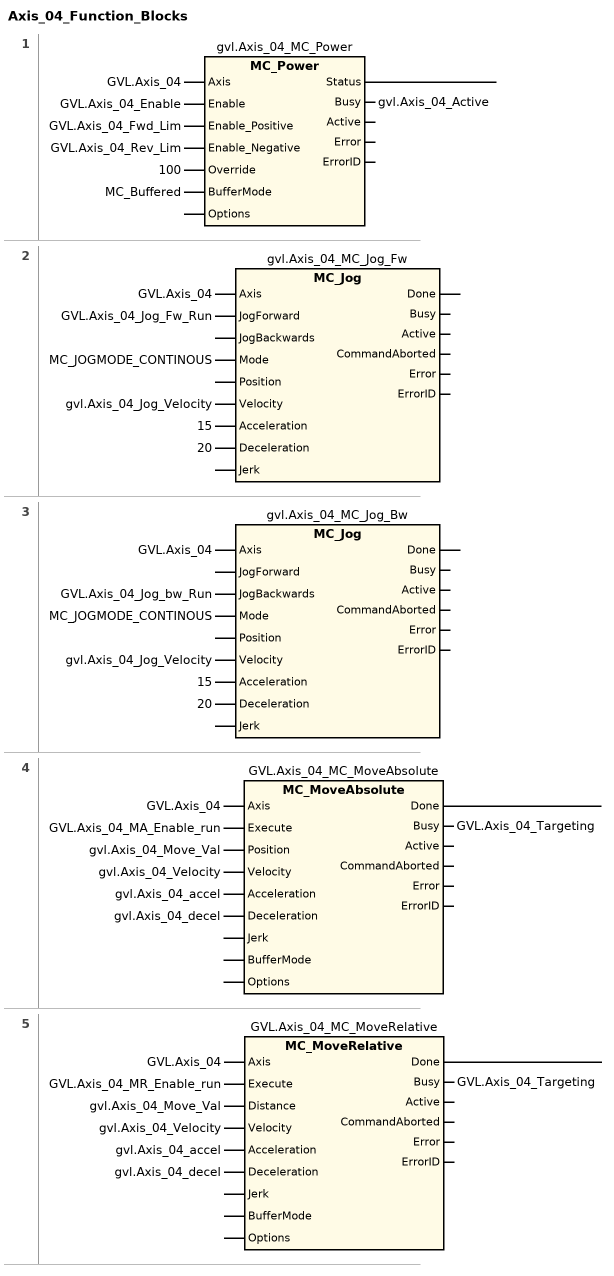
// NETWORK 1
gvl.Axis_04_MC_Power(
    Axis := GVL.Axis_04,
    Enable := GVL.Axis_04_Enable,
    Enable_Positive := GVL.Axis_04_Fwd_Lim,
    Enable_Negative := GVL.Axis_04_Rev_Lim,
    Override := 100,
    BufferMode := MC_Buffered,
    Busy => gvl.Axis_04_Active); // MC_Power

// NETWORK 2
gvl.Axis_04_MC_Jog_Fw(
    Axis := GVL.Axis_04,
    JogForward := GVL.Axis_04_Jog_Fw_Run,
    Mode := MC_JOGMODE_CONTINOUS,
    Velocity := gvl.Axis_04_Jog_Velocity,
    Acceleration := 15,
    Deceleration := 20); // MC_Jog

// NETWORK 3
gvl.Axis_04_MC_Jog_Bw(
    Axis := GVL.Axis_04,
    JogBackwards := GVL.Axis_04_Jog_bw_Run,
    Mode := MC_JOGMODE_CONTINOUS,
    Velocity := gvl.Axis_04_Jog_Velocity,
    Acceleration := 15,
    Deceleration := 20); // MC_Jog

// NETWORK 4
GVL.Axis_04_MC_MoveAbsolute(
    Axis := GVL.Axis_04,
    Execute := GVL.Axis_04_MA_Enable_run,
    Position := gvl.Axis_04_Move_Val,
    Velocity := gvl.Axis_04_Velocity,
    Acceleration := gvl.Axis_04_accel,
    Deceleration := gvl.Axis_04_decel,
    Busy => GVL.Axis_04_Targeting); // MC_MoveAbsolute

// NETWORK 5
GVL.Axis_04_MC_MoveRelative(
    Axis := GVL.Axis_04,
    Execute := GVL.Axis_04_MR_Enable_run,
    Distance := gvl.Axis_04_Move_Val,
    Velocity := gvl.Axis_04_Velocity,
    Acceleration := gvl.Axis_04_accel,
    Deceleration := gvl.Axis_04_decel,
    Busy => GVL.Axis_04_Targeting); // MC_MoveRelative

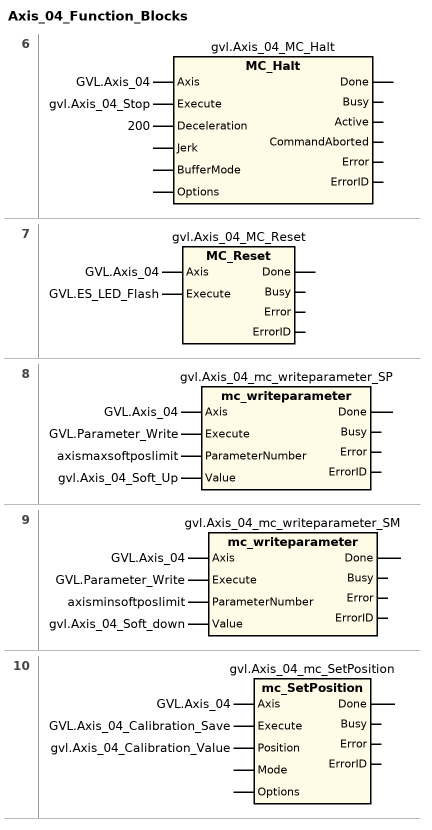
// NETWORK 6
gvl.Axis_04_MC_Halt(Axis := GVL.Axis_04, Execute := gvl.Axis_04_Stop, Deceleration := 200); // MC_Halt

// NETWORK 7
gvl.Axis_04_MC_Reset(Axis := GVL.Axis_04, Execute := GVL.ES_LED_Flash); // MC_Reset

// NETWORK 8
gvl.Axis_04_mc_writeparameter_SP(
    Axis := GVL.Axis_04,
    Execute := GVL.Parameter_Write,
    ParameterNumber := axismaxsoftposlimit,
    Value := gvl.Axis_04_Soft_Up); // mc_writeparameter

// NETWORK 9
gvl.Axis_04_mc_writeparameter_SM(
    Axis := GVL.Axis_04,
    Execute := GVL.Parameter_Write,
    ParameterNumber := axisminsoftposlimit,
    Value := gvl.Axis_04_Soft_down); // mc_writeparameter

// NETWORK 10
gvl.Axis_04_mc_SetPosition(
    Axis := GVL.Axis_04,
    Execute := GVL.Axis_04_Calibration_Save,
    Position := gvl.Axis_04_Calibration_Value); // mc_SetPosition

END_PROGRAM

// ---- POUs/Axis_04_Logic.TcPOU
PROGRAM Axis_04_Logic
VAR
	TON_0: TON;
	TON_1: TON;
	TON_2: TON;
	TON_3: TON;
	Axis_04_Velocity_Range: LREAL;
	Axis_04_Velocity_Scale: LREAL;
	Axis_04_Velocity_Raw: LREAL;
	Axis_04_Soft_Range: LREAL;
	Axis_04_Soft_Position: LREAL;
	Axis_04_Soft_Position_In_Range: LREAL;
END_VAR

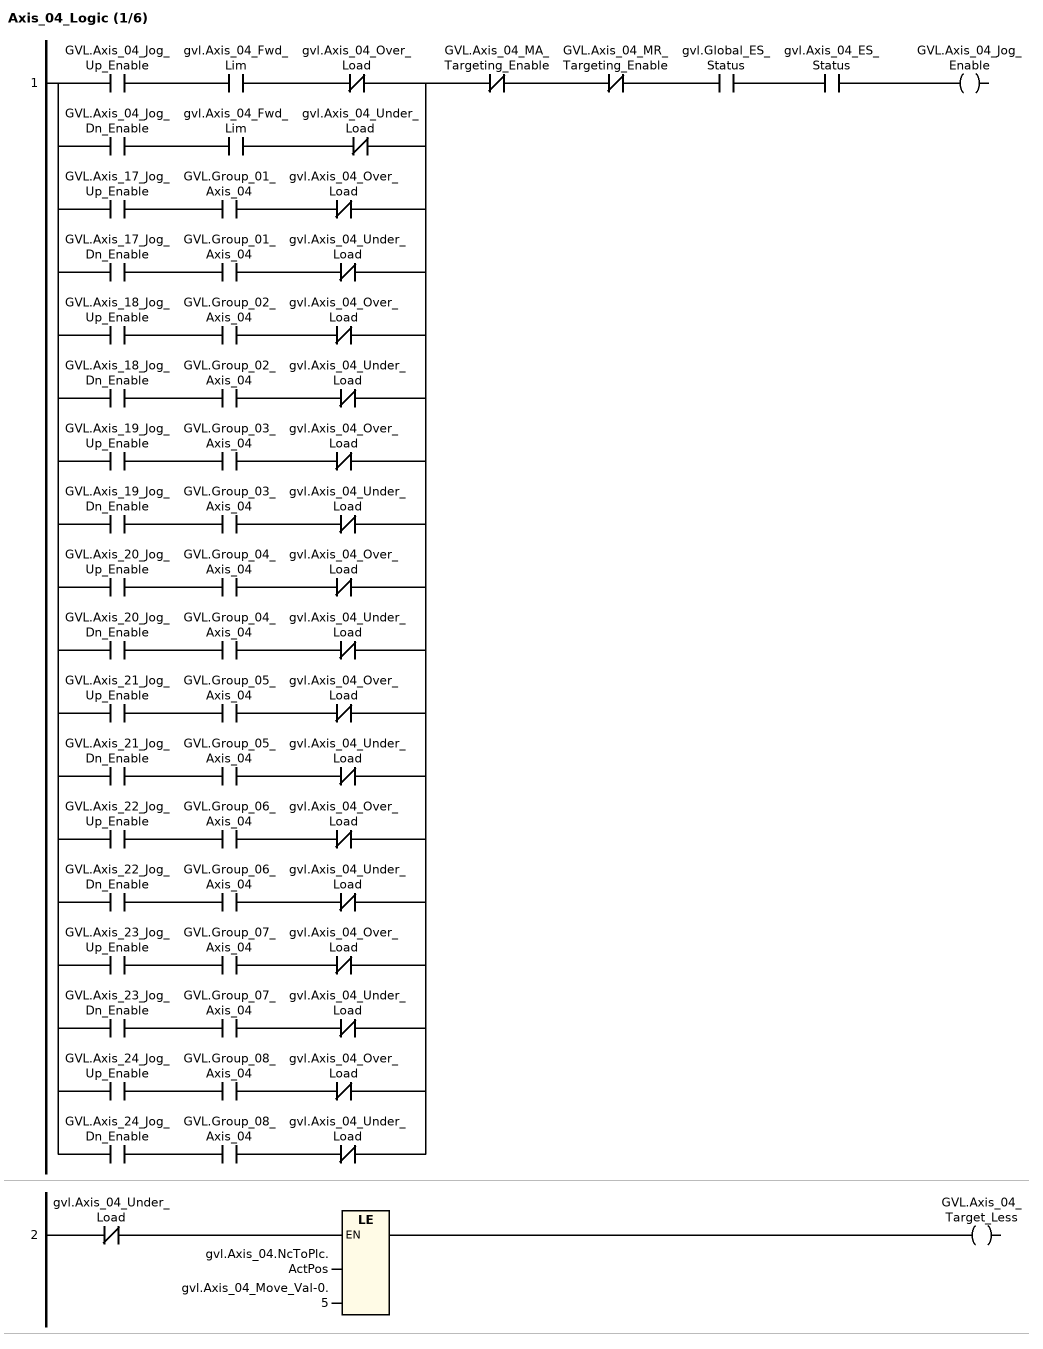
// NETWORK 1
GVL.Axis_04_Jog_Enable := (GVL.Axis_04_Jog_Up_Enable AND gvl.Axis_04_Fwd_Lim AND NOT gvl.Axis_04_Over_Load OR GVL.Axis_04_Jog_Dn_Enable AND gvl.Axis_04_Fwd_Lim AND NOT gvl.Axis_04_Under_Load OR GVL.Axis_17_Jog_Up_Enable AND GVL.Group_01_Axis_04 AND NOT gvl.Axis_04_Over_Load OR GVL.Axis_17_Jog_Dn_Enable AND GVL.Group_01_Axis_04 AND NOT gvl.Axis_04_Under_Load OR GVL.Axis_18_Jog_Up_Enable AND GVL.Group_02_Axis_04 AND NOT gvl.Axis_04_Over_Load OR GVL.Axis_18_Jog_Dn_Enable AND GVL.Group_02_Axis_04 AND NOT gvl.Axis_04_Under_Load OR GVL.Axis_19_Jog_Up_Enable AND GVL.Group_03_Axis_04 AND NOT gvl.Axis_04_Over_Load OR GVL.Axis_19_Jog_Dn_Enable AND GVL.Group_03_Axis_04 AND NOT gvl.Axis_04_Under_Load OR GVL.Axis_20_Jog_Up_Enable AND GVL.Group_04_Axis_04 AND NOT gvl.Axis_04_Over_Load OR GVL.Axis_20_Jog_Dn_Enable AND GVL.Group_04_Axis_04 AND NOT gvl.Axis_04_Under_Load OR GVL.Axis_21_Jog_Up_Enable AND GVL.Group_05_Axis_04 AND NOT gvl.Axis_04_Over_Load OR GVL.Axis_21_Jog_Dn_Enable AND GVL.Group_05_Axis_04 AND NOT gvl.Axis_04_Under_Load OR GVL.Axis_22_Jog_Up_Enable AND GVL.Group_06_Axis_04 AND NOT gvl.Axis_04_Over_Load OR GVL.Axis_22_Jog_Dn_Enable AND GVL.Group_06_Axis_04 AND NOT gvl.Axis_04_Under_Load OR GVL.Axis_23_Jog_Up_Enable AND GVL.Group_07_Axis_04 AND NOT gvl.Axis_04_Over_Load OR GVL.Axis_23_Jog_Dn_Enable AND GVL.Group_07_Axis_04 AND NOT gvl.Axis_04_Under_Load OR GVL.Axis_24_Jog_Up_Enable AND GVL.Group_08_Axis_04 AND NOT gvl.Axis_04_Over_Load OR GVL.Axis_24_Jog_Dn_Enable AND GVL.Group_08_Axis_04 AND NOT gvl.Axis_04_Under_Load) AND NOT GVL.Axis_04_MA_Targeting_Enable AND NOT GVL.Axis_04_MR_Targeting_Enable AND gvl.Global_ES_Status AND gvl.Axis_04_ES_Status;

// NETWORK 2
GVL.Axis_04_Target_Less := NOT gvl.Axis_04_Under_Load AND gvl.Axis_04.NcToPlc.ActPos <= (gvl.Axis_04_Move_Val-0.5);

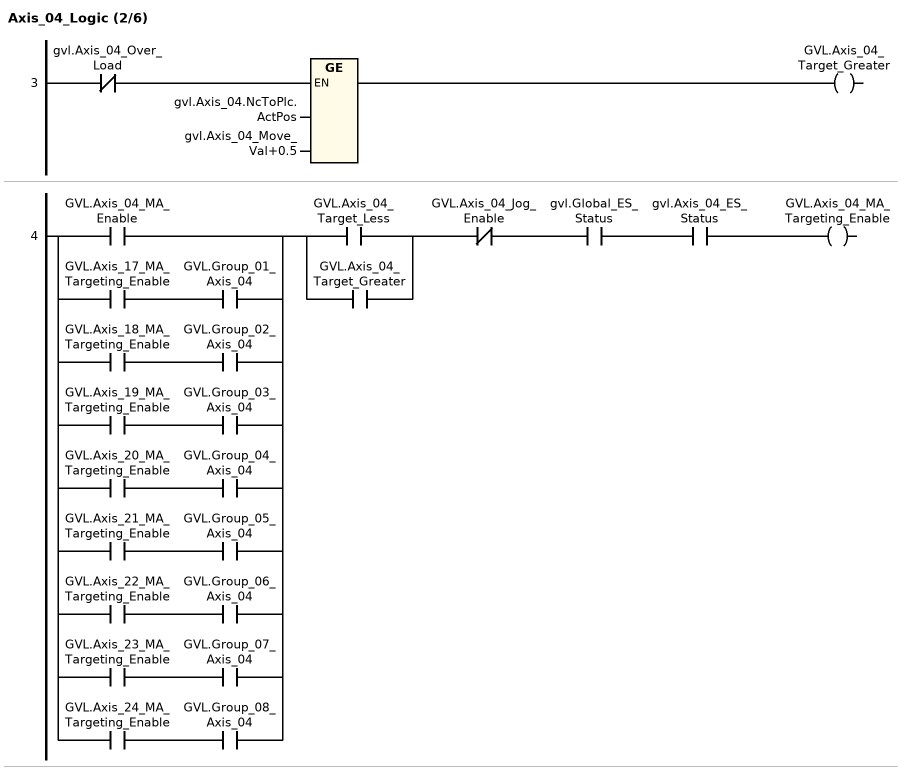
// NETWORK 3
GVL.Axis_04_Target_Greater := NOT gvl.Axis_04_Over_Load AND gvl.Axis_04.NcToPlc.ActPos >= (gvl.Axis_04_Move_Val+0.5);

// NETWORK 4
GVL.Axis_04_MA_Targeting_Enable := (GVL.Axis_04_MA_Enable OR GVL.Axis_17_MA_Targeting_Enable AND GVL.Group_01_Axis_04 OR GVL.Axis_18_MA_Targeting_Enable AND GVL.Group_02_Axis_04 OR GVL.Axis_19_MA_Targeting_Enable AND GVL.Group_03_Axis_04 OR GVL.Axis_20_MA_Targeting_Enable AND GVL.Group_04_Axis_04 OR GVL.Axis_21_MA_Targeting_Enable AND GVL.Group_05_Axis_04 OR GVL.Axis_22_MA_Targeting_Enable AND GVL.Group_06_Axis_04 OR GVL.Axis_23_MA_Targeting_Enable AND GVL.Group_07_Axis_04 OR GVL.Axis_24_MA_Targeting_Enable AND GVL.Group_08_Axis_04) AND (GVL.Axis_04_Target_Less OR GVL.Axis_04_Target_Greater) AND NOT GVL.Axis_04_Jog_Enable AND gvl.Global_ES_Status AND gvl.Axis_04_ES_Status;

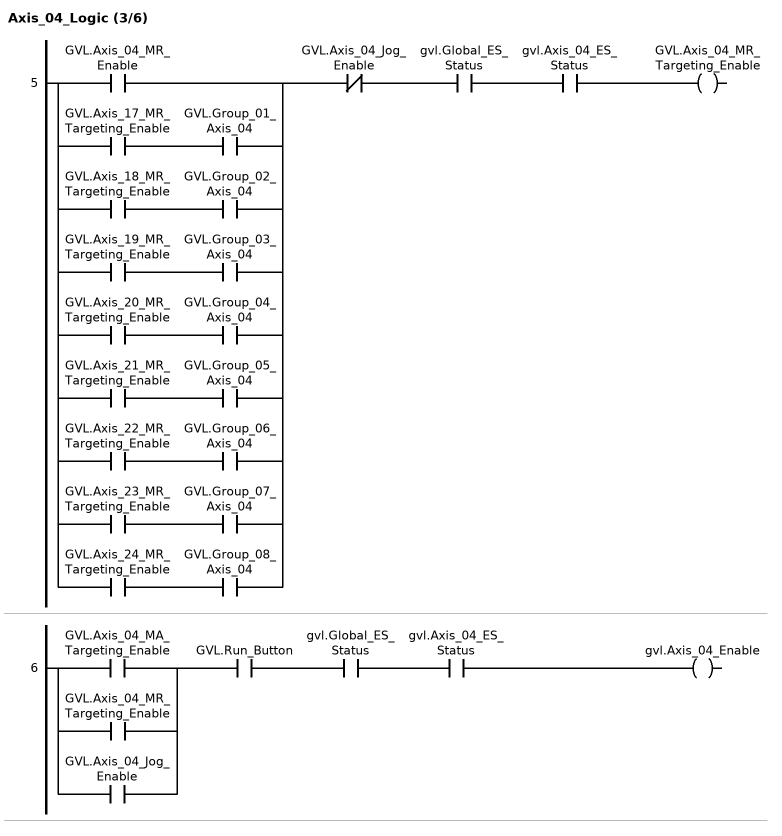
// NETWORK 5
GVL.Axis_04_MR_Targeting_Enable := (GVL.Axis_04_MR_Enable OR GVL.Axis_17_MR_Targeting_Enable AND GVL.Group_01_Axis_04 OR GVL.Axis_18_MR_Targeting_Enable AND GVL.Group_02_Axis_04 OR GVL.Axis_19_MR_Targeting_Enable AND GVL.Group_03_Axis_04 OR GVL.Axis_20_MR_Targeting_Enable AND GVL.Group_04_Axis_04 OR GVL.Axis_21_MR_Targeting_Enable AND GVL.Group_05_Axis_04 OR GVL.Axis_22_MR_Targeting_Enable AND GVL.Group_06_Axis_04 OR GVL.Axis_23_MR_Targeting_Enable AND GVL.Group_07_Axis_04 OR GVL.Axis_24_MR_Targeting_Enable AND GVL.Group_08_Axis_04) AND NOT GVL.Axis_04_Jog_Enable AND gvl.Global_ES_Status AND gvl.Axis_04_ES_Status;

// NETWORK 6
gvl.Axis_04_Enable := (GVL.Axis_04_MA_Targeting_Enable OR GVL.Axis_04_MR_Targeting_Enable OR GVL.Axis_04_Jog_Enable) AND GVL.Run_Button AND gvl.Global_ES_Status AND gvl.Axis_04_ES_Status;

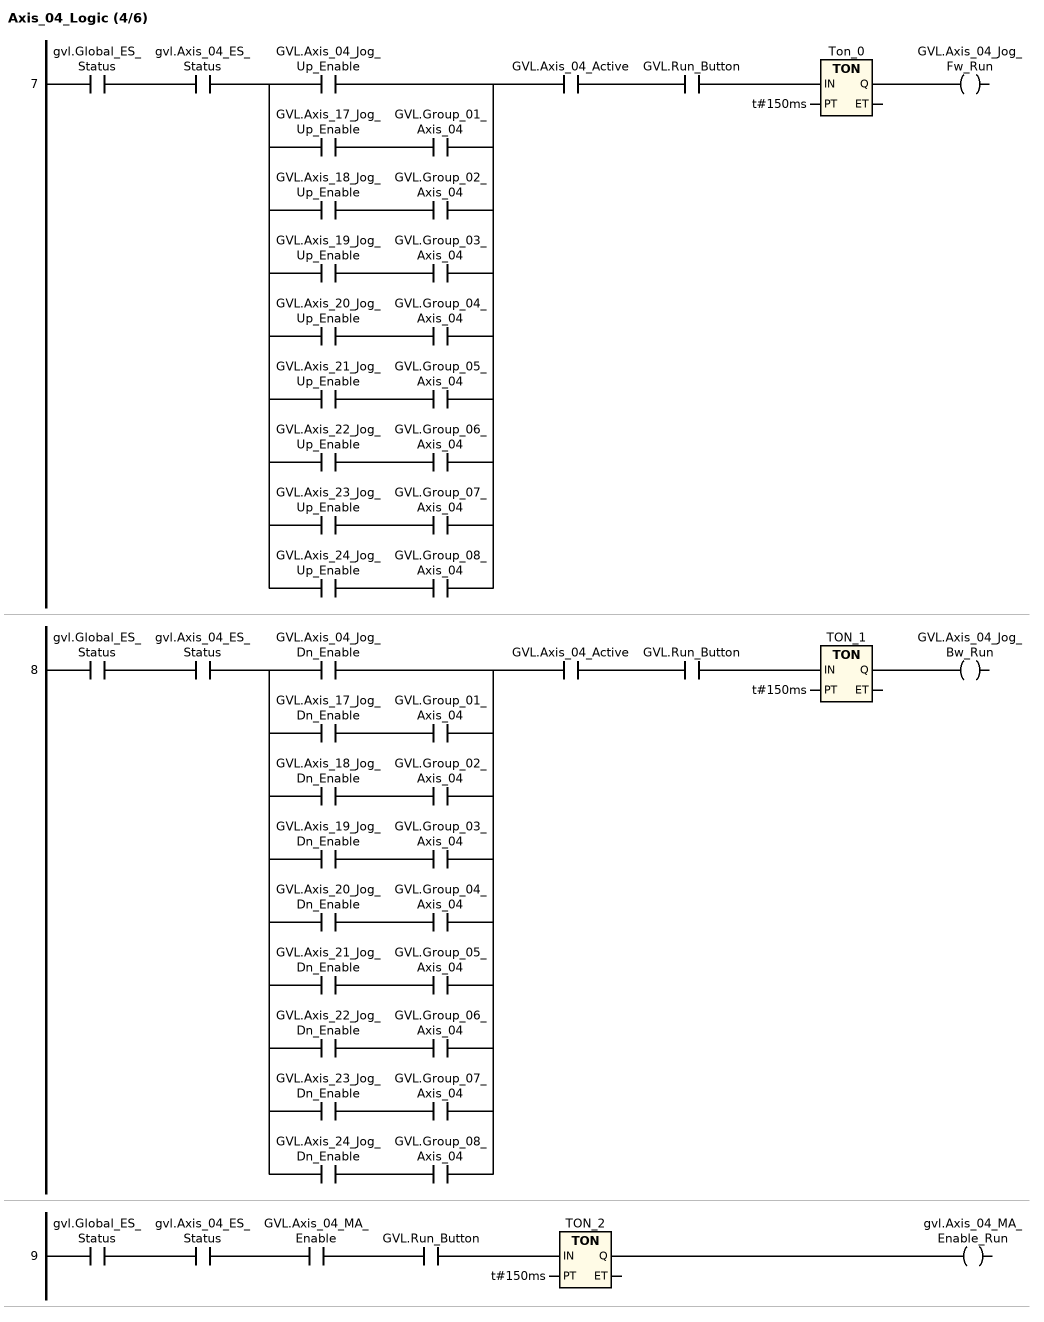
// NETWORK 7
Ton_0(IN := gvl.Global_ES_Status AND gvl.Axis_04_ES_Status AND (GVL.Axis_04_Jog_Up_Enable OR GVL.Axis_17_Jog_Up_Enable AND GVL.Group_01_Axis_04 OR GVL.Axis_18_Jog_Up_Enable AND GVL.Group_02_Axis_04 OR GVL.Axis_19_Jog_Up_Enable AND GVL.Group_03_Axis_04 OR GVL.Axis_20_Jog_Up_Enable AND GVL.Group_04_Axis_04 OR GVL.Axis_21_Jog_Up_Enable AND GVL.Group_05_Axis_04 OR GVL.Axis_22_Jog_Up_Enable AND GVL.Group_06_Axis_04 OR GVL.Axis_23_Jog_Up_Enable AND GVL.Group_07_Axis_04 OR GVL.Axis_24_Jog_Up_Enable AND GVL.Group_08_Axis_04) AND GVL.Axis_04_Active AND GVL.Run_Button, PT := t#150ms); // TON
GVL.Axis_04_Jog_Fw_Run := Ton_0.Q;

// NETWORK 8
TON_1(IN := gvl.Global_ES_Status AND gvl.Axis_04_ES_Status AND (GVL.Axis_04_Jog_Dn_Enable OR GVL.Axis_17_Jog_Dn_Enable AND GVL.Group_01_Axis_04 OR GVL.Axis_18_Jog_Dn_Enable AND GVL.Group_02_Axis_04 OR GVL.Axis_19_Jog_Dn_Enable AND GVL.Group_03_Axis_04 OR GVL.Axis_20_Jog_Dn_Enable AND GVL.Group_04_Axis_04 OR GVL.Axis_21_Jog_Dn_Enable AND GVL.Group_05_Axis_04 OR GVL.Axis_22_Jog_Dn_Enable AND GVL.Group_06_Axis_04 OR GVL.Axis_23_Jog_Dn_Enable AND GVL.Group_07_Axis_04 OR GVL.Axis_24_Jog_Dn_Enable AND GVL.Group_08_Axis_04) AND GVL.Axis_04_Active AND GVL.Run_Button, PT := t#150ms); // TON
GVL.Axis_04_Jog_Bw_Run := TON_1.Q;

// NETWORK 9
TON_2(IN := gvl.Global_ES_Status AND gvl.Axis_04_ES_Status AND GVL.Axis_04_MA_Enable AND GVL.Run_Button, PT := t#150ms); // TON
gvl.Axis_04_MA_Enable_Run := TON_2.Q;

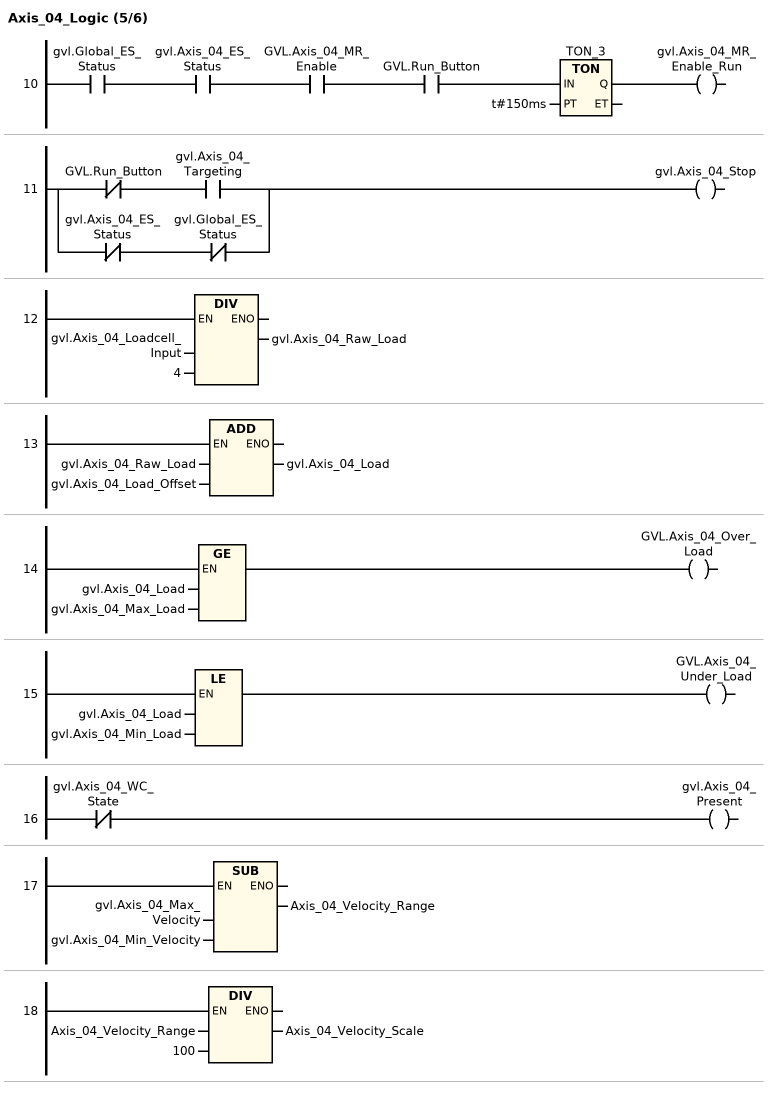
// NETWORK 10
TON_3(IN := gvl.Global_ES_Status AND gvl.Axis_04_ES_Status AND GVL.Axis_04_MR_Enable AND GVL.Run_Button, PT := t#150ms); // TON
gvl.Axis_04_MR_Enable_Run := TON_3.Q;

// NETWORK 11
gvl.Axis_04_Stop := NOT GVL.Run_Button AND gvl.Axis_04_Targeting OR NOT gvl.Axis_04_ES_Status AND NOT gvl.Global_ES_Status;

// NETWORK 12
gvl.Axis_04_Raw_Load := gvl.Axis_04_Loadcell_Input / 4;

// NETWORK 13
gvl.Axis_04_Load := gvl.Axis_04_Raw_Load + gvl.Axis_04_Load_Offset;

// NETWORK 14
GVL.Axis_04_Over_Load := gvl.Axis_04_Load >= gvl.Axis_04_Max_Load;

// NETWORK 15
GVL.Axis_04_Under_Load := gvl.Axis_04_Load <= gvl.Axis_04_Min_Load;

// NETWORK 16
gvl.Axis_04_Present := NOT gvl.Axis_04_WC_State;

// NETWORK 17
Axis_04_Velocity_Range := gvl.Axis_04_Max_Velocity - gvl.Axis_04_Min_Velocity;

// NETWORK 18
Axis_04_Velocity_Scale := Axis_04_Velocity_Range / 100;

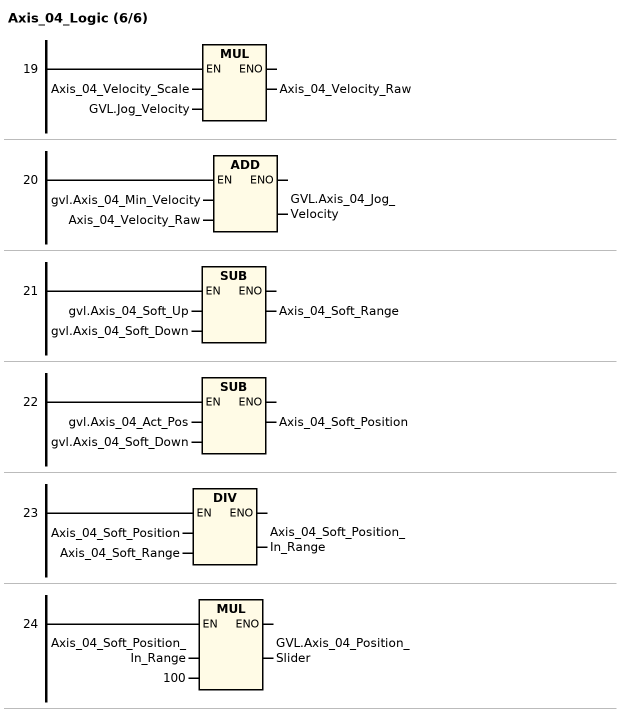
// NETWORK 19
Axis_04_Velocity_Raw := Axis_04_Velocity_Scale * GVL.Jog_Velocity;

// NETWORK 20
GVL.Axis_04_Jog_Velocity := gvl.Axis_04_Min_Velocity + Axis_04_Velocity_Raw;

// NETWORK 21
Axis_04_Soft_Range := gvl.Axis_04_Soft_Up - gvl.Axis_04_Soft_Down;

// NETWORK 22
Axis_04_Soft_Position := gvl.Axis_04_Act_Pos - gvl.Axis_04_Soft_Down;

// NETWORK 23
Axis_04_Soft_Position_In_Range := Axis_04_Soft_Position / Axis_04_Soft_Range;

// NETWORK 24
GVL.Axis_04_Position_Slider := Axis_04_Soft_Position_In_Range * 100;

END_PROGRAM

// ---- POUs/Axis_05_Function_Blocks.TcPOU
PROGRAM Axis_05_Function_Blocks
VAR
END_VAR

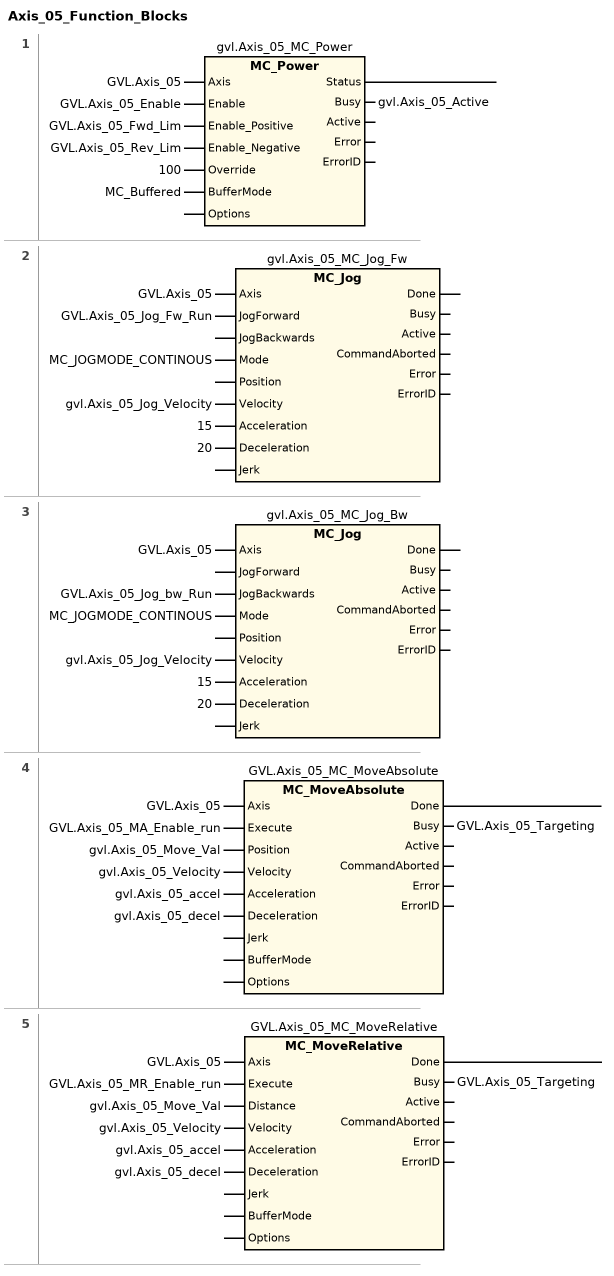
// NETWORK 1
gvl.Axis_05_MC_Power(
    Axis := GVL.Axis_05,
    Enable := GVL.Axis_05_Enable,
    Enable_Positive := GVL.Axis_05_Fwd_Lim,
    Enable_Negative := GVL.Axis_05_Rev_Lim,
    Override := 100,
    BufferMode := MC_Buffered,
    Busy => gvl.Axis_05_Active); // MC_Power

// NETWORK 2
gvl.Axis_05_MC_Jog_Fw(
    Axis := GVL.Axis_05,
    JogForward := GVL.Axis_05_Jog_Fw_Run,
    Mode := MC_JOGMODE_CONTINOUS,
    Velocity := gvl.Axis_05_Jog_Velocity,
    Acceleration := 15,
    Deceleration := 20); // MC_Jog

// NETWORK 3
gvl.Axis_05_MC_Jog_Bw(
    Axis := GVL.Axis_05,
    JogBackwards := GVL.Axis_05_Jog_bw_Run,
    Mode := MC_JOGMODE_CONTINOUS,
    Velocity := gvl.Axis_05_Jog_Velocity,
    Acceleration := 15,
    Deceleration := 20); // MC_Jog

// NETWORK 4
GVL.Axis_05_MC_MoveAbsolute(
    Axis := GVL.Axis_05,
    Execute := GVL.Axis_05_MA_Enable_run,
    Position := gvl.Axis_05_Move_Val,
    Velocity := gvl.Axis_05_Velocity,
    Acceleration := gvl.Axis_05_accel,
    Deceleration := gvl.Axis_05_decel,
    Busy => GVL.Axis_05_Targeting); // MC_MoveAbsolute

// NETWORK 5
GVL.Axis_05_MC_MoveRelative(
    Axis := GVL.Axis_05,
    Execute := GVL.Axis_05_MR_Enable_run,
    Distance := gvl.Axis_05_Move_Val,
    Velocity := gvl.Axis_05_Velocity,
    Acceleration := gvl.Axis_05_accel,
    Deceleration := gvl.Axis_05_decel,
    Busy => GVL.Axis_05_Targeting); // MC_MoveRelative

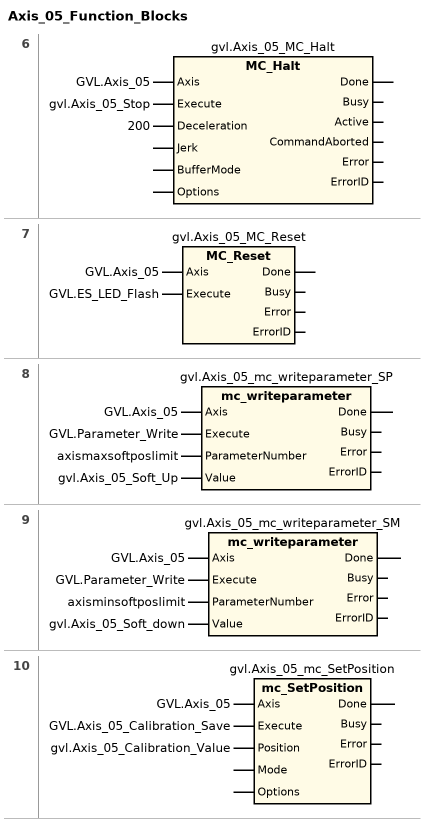
// NETWORK 6
gvl.Axis_05_MC_Halt(Axis := GVL.Axis_05, Execute := gvl.Axis_05_Stop, Deceleration := 200); // MC_Halt

// NETWORK 7
gvl.Axis_05_MC_Reset(Axis := GVL.Axis_05, Execute := GVL.ES_LED_Flash); // MC_Reset

// NETWORK 8
gvl.Axis_05_mc_writeparameter_SP(
    Axis := GVL.Axis_05,
    Execute := GVL.Parameter_Write,
    ParameterNumber := axismaxsoftposlimit,
    Value := gvl.Axis_05_Soft_Up); // mc_writeparameter

// NETWORK 9
gvl.Axis_05_mc_writeparameter_SM(
    Axis := GVL.Axis_05,
    Execute := GVL.Parameter_Write,
    ParameterNumber := axisminsoftposlimit,
    Value := gvl.Axis_05_Soft_down); // mc_writeparameter

// NETWORK 10
gvl.Axis_05_mc_SetPosition(
    Axis := GVL.Axis_05,
    Execute := GVL.Axis_05_Calibration_Save,
    Position := gvl.Axis_05_Calibration_Value); // mc_SetPosition

END_PROGRAM

// ---- POUs/Axis_05_Logic.TcPOU
PROGRAM Axis_05_Logic
VAR
	TON_0: TON;
	TON_1: TON;
	TON_2: TON;
	TON_3: TON;
	Axis_05_Velocity_Range: LREAL;
	Axis_05_Velocity_Scale: LREAL;
	Axis_05_Velocity_Raw: LREAL;
	Axis_05_Soft_Range: LREAL;
	Axis_05_Soft_Position: LREAL;
	Axis_05_Soft_Position_In_Range: LREAL;
END_VAR

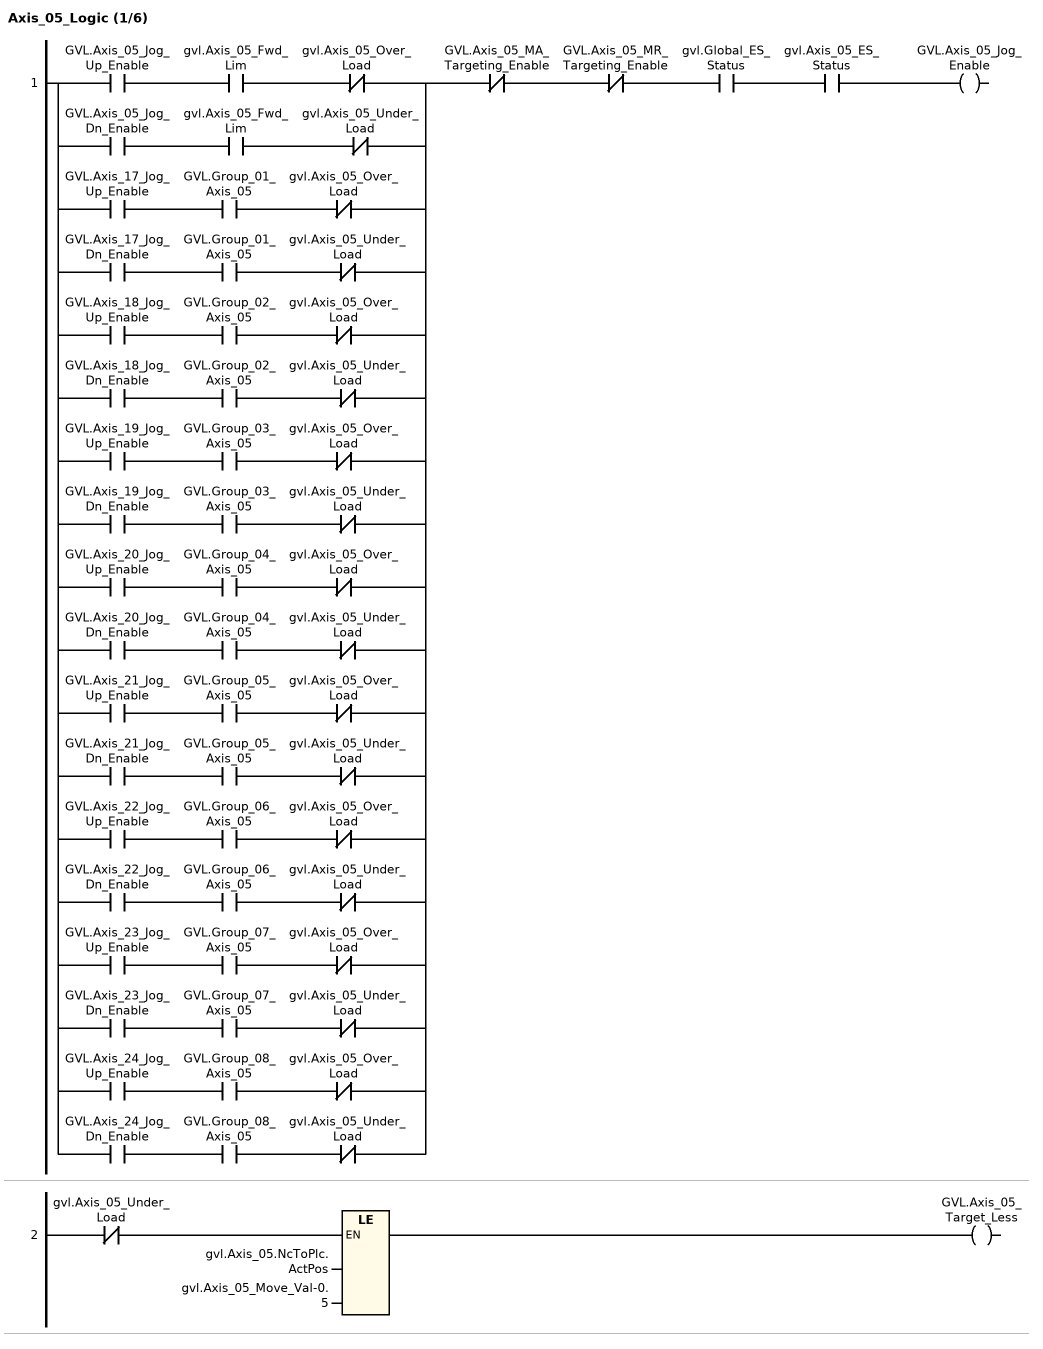
// NETWORK 1
GVL.Axis_05_Jog_Enable := (GVL.Axis_05_Jog_Up_Enable AND gvl.Axis_05_Fwd_Lim AND NOT gvl.Axis_05_Over_Load OR GVL.Axis_05_Jog_Dn_Enable AND gvl.Axis_05_Fwd_Lim AND NOT gvl.Axis_05_Under_Load OR GVL.Axis_17_Jog_Up_Enable AND GVL.Group_01_Axis_05 AND NOT gvl.Axis_05_Over_Load OR GVL.Axis_17_Jog_Dn_Enable AND GVL.Group_01_Axis_05 AND NOT gvl.Axis_05_Under_Load OR GVL.Axis_18_Jog_Up_Enable AND GVL.Group_02_Axis_05 AND NOT gvl.Axis_05_Over_Load OR GVL.Axis_18_Jog_Dn_Enable AND GVL.Group_02_Axis_05 AND NOT gvl.Axis_05_Under_Load OR GVL.Axis_19_Jog_Up_Enable AND GVL.Group_03_Axis_05 AND NOT gvl.Axis_05_Over_Load OR GVL.Axis_19_Jog_Dn_Enable AND GVL.Group_03_Axis_05 AND NOT gvl.Axis_05_Under_Load OR GVL.Axis_20_Jog_Up_Enable AND GVL.Group_04_Axis_05 AND NOT gvl.Axis_05_Over_Load OR GVL.Axis_20_Jog_Dn_Enable AND GVL.Group_04_Axis_05 AND NOT gvl.Axis_05_Under_Load OR GVL.Axis_21_Jog_Up_Enable AND GVL.Group_05_Axis_05 AND NOT gvl.Axis_05_Over_Load OR GVL.Axis_21_Jog_Dn_Enable AND GVL.Group_05_Axis_05 AND NOT gvl.Axis_05_Under_Load OR GVL.Axis_22_Jog_Up_Enable AND GVL.Group_06_Axis_05 AND NOT gvl.Axis_05_Over_Load OR GVL.Axis_22_Jog_Dn_Enable AND GVL.Group_06_Axis_05 AND NOT gvl.Axis_05_Under_Load OR GVL.Axis_23_Jog_Up_Enable AND GVL.Group_07_Axis_05 AND NOT gvl.Axis_05_Over_Load OR GVL.Axis_23_Jog_Dn_Enable AND GVL.Group_07_Axis_05 AND NOT gvl.Axis_05_Under_Load OR GVL.Axis_24_Jog_Up_Enable AND GVL.Group_08_Axis_05 AND NOT gvl.Axis_05_Over_Load OR GVL.Axis_24_Jog_Dn_Enable AND GVL.Group_08_Axis_05 AND NOT gvl.Axis_05_Under_Load) AND NOT GVL.Axis_05_MA_Targeting_Enable AND NOT GVL.Axis_05_MR_Targeting_Enable AND gvl.Global_ES_Status AND gvl.Axis_05_ES_Status;

// NETWORK 2
GVL.Axis_05_Target_Less := NOT gvl.Axis_05_Under_Load AND gvl.Axis_05.NcToPlc.ActPos <= (gvl.Axis_05_Move_Val-0.5);

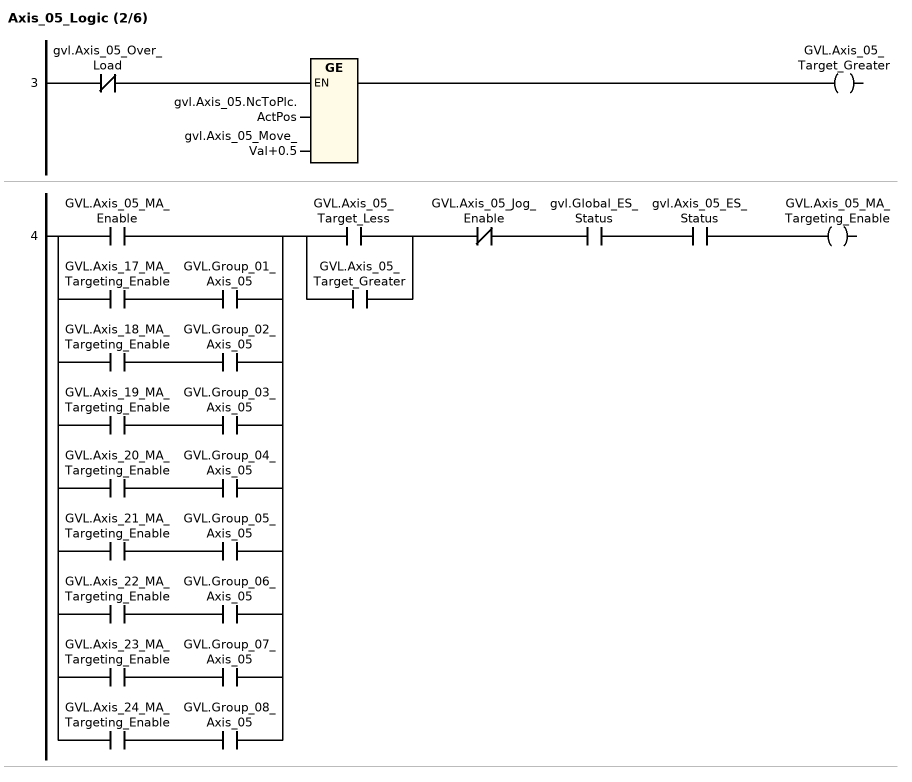
// NETWORK 3
GVL.Axis_05_Target_Greater := NOT gvl.Axis_05_Over_Load AND gvl.Axis_05.NcToPlc.ActPos >= (gvl.Axis_05_Move_Val+0.5);

// NETWORK 4
GVL.Axis_05_MA_Targeting_Enable := (GVL.Axis_05_MA_Enable OR GVL.Axis_17_MA_Targeting_Enable AND GVL.Group_01_Axis_05 OR GVL.Axis_18_MA_Targeting_Enable AND GVL.Group_02_Axis_05 OR GVL.Axis_19_MA_Targeting_Enable AND GVL.Group_03_Axis_05 OR GVL.Axis_20_MA_Targeting_Enable AND GVL.Group_04_Axis_05 OR GVL.Axis_21_MA_Targeting_Enable AND GVL.Group_05_Axis_05 OR GVL.Axis_22_MA_Targeting_Enable AND GVL.Group_06_Axis_05 OR GVL.Axis_23_MA_Targeting_Enable AND GVL.Group_07_Axis_05 OR GVL.Axis_24_MA_Targeting_Enable AND GVL.Group_08_Axis_05) AND (GVL.Axis_05_Target_Less OR GVL.Axis_05_Target_Greater) AND NOT GVL.Axis_05_Jog_Enable AND gvl.Global_ES_Status AND gvl.Axis_05_ES_Status;

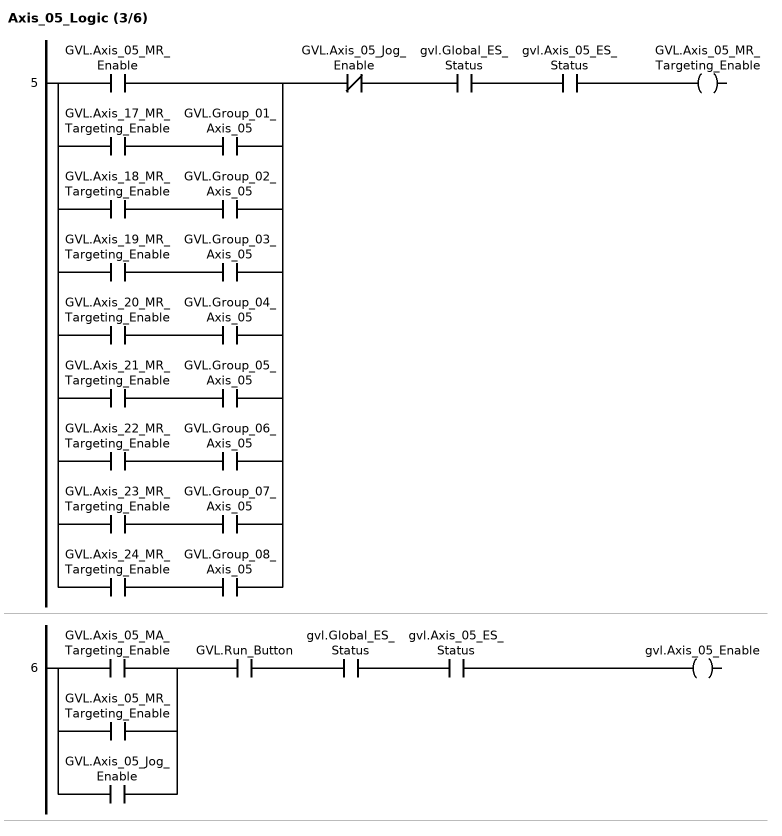
// NETWORK 5
GVL.Axis_05_MR_Targeting_Enable := (GVL.Axis_05_MR_Enable OR GVL.Axis_17_MR_Targeting_Enable AND GVL.Group_01_Axis_05 OR GVL.Axis_18_MR_Targeting_Enable AND GVL.Group_02_Axis_05 OR GVL.Axis_19_MR_Targeting_Enable AND GVL.Group_03_Axis_05 OR GVL.Axis_20_MR_Targeting_Enable AND GVL.Group_04_Axis_05 OR GVL.Axis_21_MR_Targeting_Enable AND GVL.Group_05_Axis_05 OR GVL.Axis_22_MR_Targeting_Enable AND GVL.Group_06_Axis_05 OR GVL.Axis_23_MR_Targeting_Enable AND GVL.Group_07_Axis_05 OR GVL.Axis_24_MR_Targeting_Enable AND GVL.Group_08_Axis_05) AND NOT GVL.Axis_05_Jog_Enable AND gvl.Global_ES_Status AND gvl.Axis_05_ES_Status;

// NETWORK 6
gvl.Axis_05_Enable := (GVL.Axis_05_MA_Targeting_Enable OR GVL.Axis_05_MR_Targeting_Enable OR GVL.Axis_05_Jog_Enable) AND GVL.Run_Button AND gvl.Global_ES_Status AND gvl.Axis_05_ES_Status;

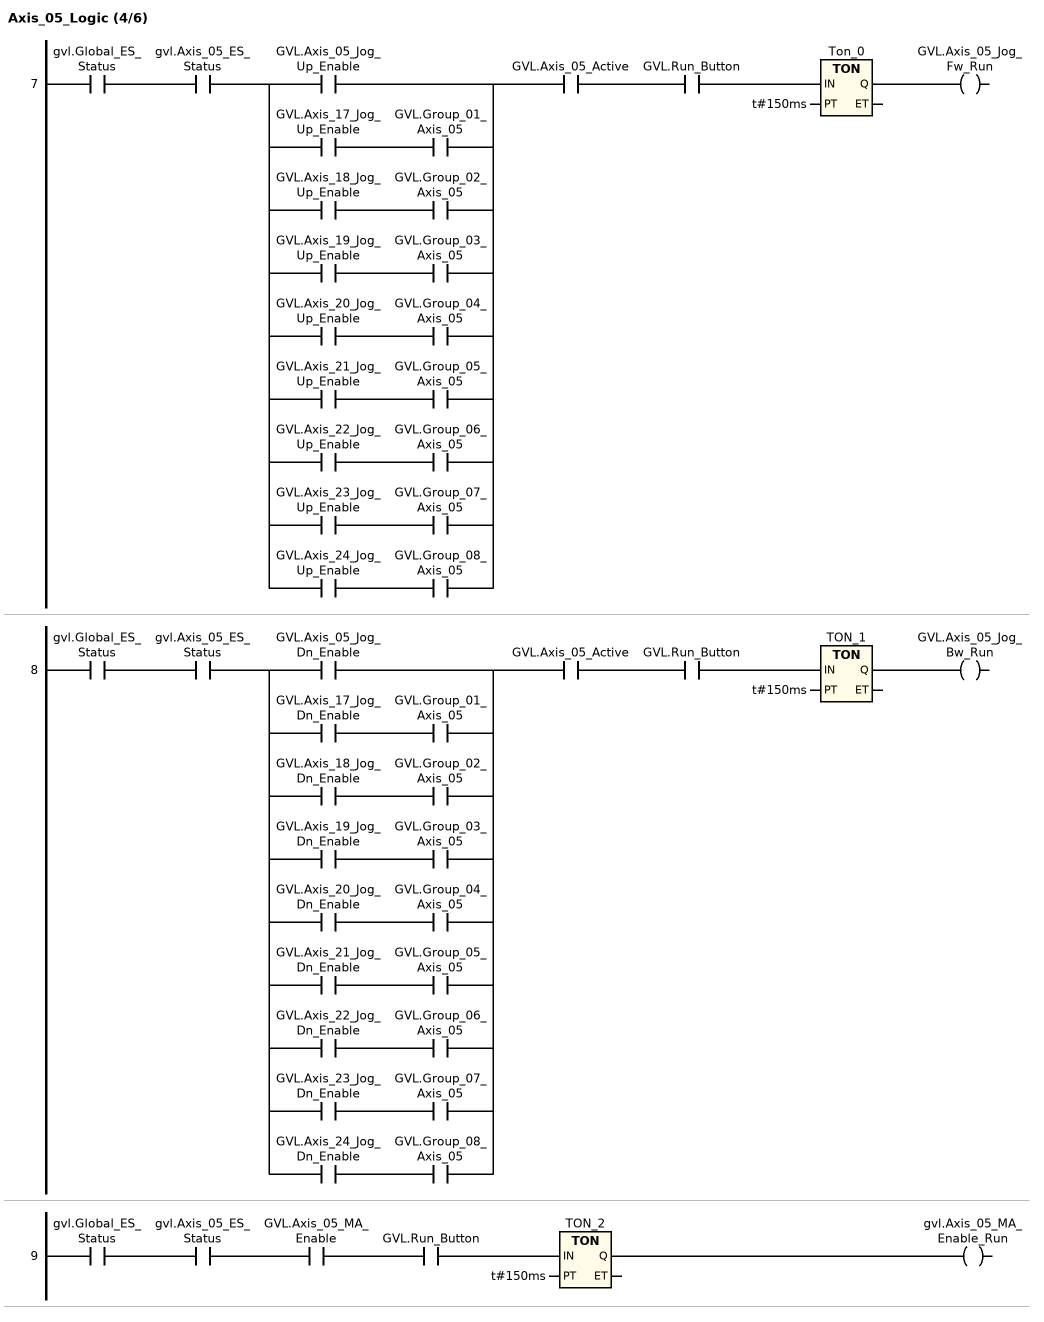
// NETWORK 7
Ton_0(IN := gvl.Global_ES_Status AND gvl.Axis_05_ES_Status AND (GVL.Axis_05_Jog_Up_Enable OR GVL.Axis_17_Jog_Up_Enable AND GVL.Group_01_Axis_05 OR GVL.Axis_18_Jog_Up_Enable AND GVL.Group_02_Axis_05 OR GVL.Axis_19_Jog_Up_Enable AND GVL.Group_03_Axis_05 OR GVL.Axis_20_Jog_Up_Enable AND GVL.Group_04_Axis_05 OR GVL.Axis_21_Jog_Up_Enable AND GVL.Group_05_Axis_05 OR GVL.Axis_22_Jog_Up_Enable AND GVL.Group_06_Axis_05 OR GVL.Axis_23_Jog_Up_Enable AND GVL.Group_07_Axis_05 OR GVL.Axis_24_Jog_Up_Enable AND GVL.Group_08_Axis_05) AND GVL.Axis_05_Active AND GVL.Run_Button, PT := t#150ms); // TON
GVL.Axis_05_Jog_Fw_Run := Ton_0.Q;

// NETWORK 8
TON_1(IN := gvl.Global_ES_Status AND gvl.Axis_05_ES_Status AND (GVL.Axis_05_Jog_Dn_Enable OR GVL.Axis_17_Jog_Dn_Enable AND GVL.Group_01_Axis_05 OR GVL.Axis_18_Jog_Dn_Enable AND GVL.Group_02_Axis_05 OR GVL.Axis_19_Jog_Dn_Enable AND GVL.Group_03_Axis_05 OR GVL.Axis_20_Jog_Dn_Enable AND GVL.Group_04_Axis_05 OR GVL.Axis_21_Jog_Dn_Enable AND GVL.Group_05_Axis_05 OR GVL.Axis_22_Jog_Dn_Enable AND GVL.Group_06_Axis_05 OR GVL.Axis_23_Jog_Dn_Enable AND GVL.Group_07_Axis_05 OR GVL.Axis_24_Jog_Dn_Enable AND GVL.Group_08_Axis_05) AND GVL.Axis_05_Active AND GVL.Run_Button, PT := t#150ms); // TON
GVL.Axis_05_Jog_Bw_Run := TON_1.Q;

// NETWORK 9
TON_2(IN := gvl.Global_ES_Status AND gvl.Axis_05_ES_Status AND GVL.Axis_05_MA_Enable AND GVL.Run_Button, PT := t#150ms); // TON
gvl.Axis_05_MA_Enable_Run := TON_2.Q;

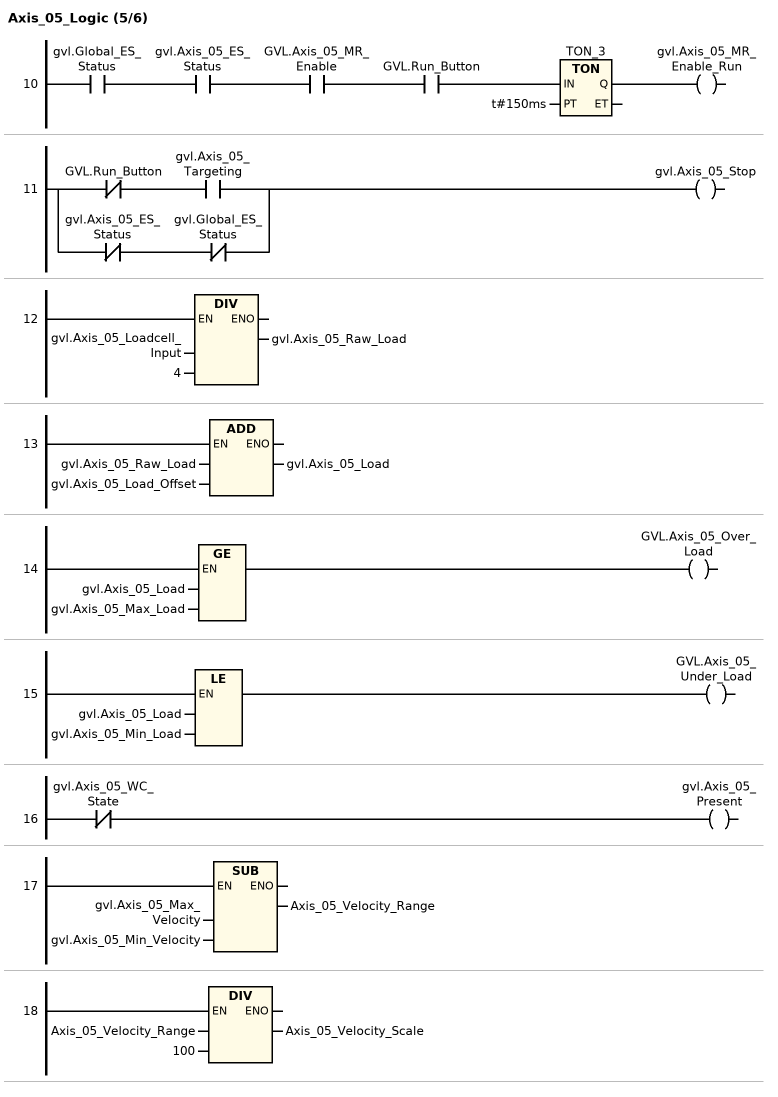
// NETWORK 10
TON_3(IN := gvl.Global_ES_Status AND gvl.Axis_05_ES_Status AND GVL.Axis_05_MR_Enable AND GVL.Run_Button, PT := t#150ms); // TON
gvl.Axis_05_MR_Enable_Run := TON_3.Q;

// NETWORK 11
gvl.Axis_05_Stop := NOT GVL.Run_Button AND gvl.Axis_05_Targeting OR NOT gvl.Axis_05_ES_Status AND NOT gvl.Global_ES_Status;

// NETWORK 12
gvl.Axis_05_Raw_Load := gvl.Axis_05_Loadcell_Input / 4;

// NETWORK 13
gvl.Axis_05_Load := gvl.Axis_05_Raw_Load + gvl.Axis_05_Load_Offset;

// NETWORK 14
GVL.Axis_05_Over_Load := gvl.Axis_05_Load >= gvl.Axis_05_Max_Load;

// NETWORK 15
GVL.Axis_05_Under_Load := gvl.Axis_05_Load <= gvl.Axis_05_Min_Load;

// NETWORK 16
gvl.Axis_05_Present := NOT gvl.Axis_05_WC_State;

// NETWORK 17
Axis_05_Velocity_Range := gvl.Axis_05_Max_Velocity - gvl.Axis_05_Min_Velocity;

// NETWORK 18
Axis_05_Velocity_Scale := Axis_05_Velocity_Range / 100;

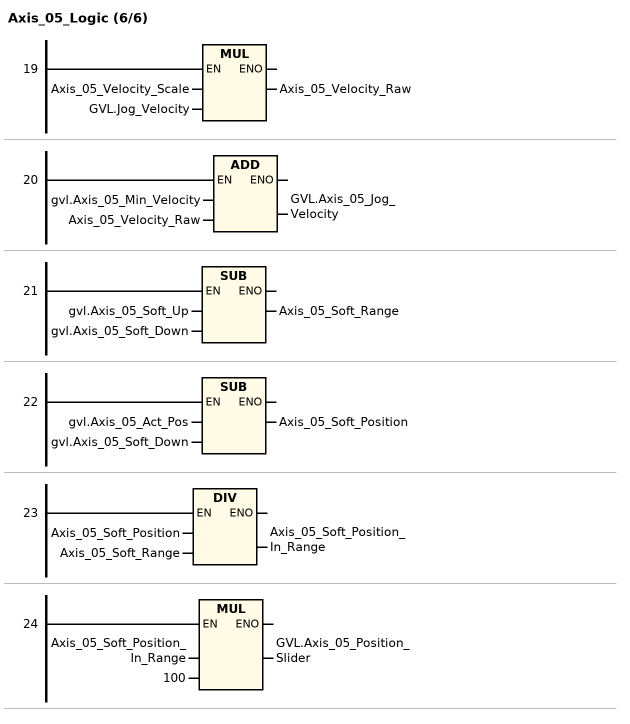
// NETWORK 19
Axis_05_Velocity_Raw := Axis_05_Velocity_Scale * GVL.Jog_Velocity;

// NETWORK 20
GVL.Axis_05_Jog_Velocity := gvl.Axis_05_Min_Velocity + Axis_05_Velocity_Raw;

// NETWORK 21
Axis_05_Soft_Range := gvl.Axis_05_Soft_Up - gvl.Axis_05_Soft_Down;

// NETWORK 22
Axis_05_Soft_Position := gvl.Axis_05_Act_Pos - gvl.Axis_05_Soft_Down;

// NETWORK 23
Axis_05_Soft_Position_In_Range := Axis_05_Soft_Position / Axis_05_Soft_Range;

// NETWORK 24
GVL.Axis_05_Position_Slider := Axis_05_Soft_Position_In_Range * 100;

END_PROGRAM

// ---- POUs/Axis_06_Function_Blocks.TcPOU
PROGRAM Axis_06_Function_Blocks
VAR
END_VAR

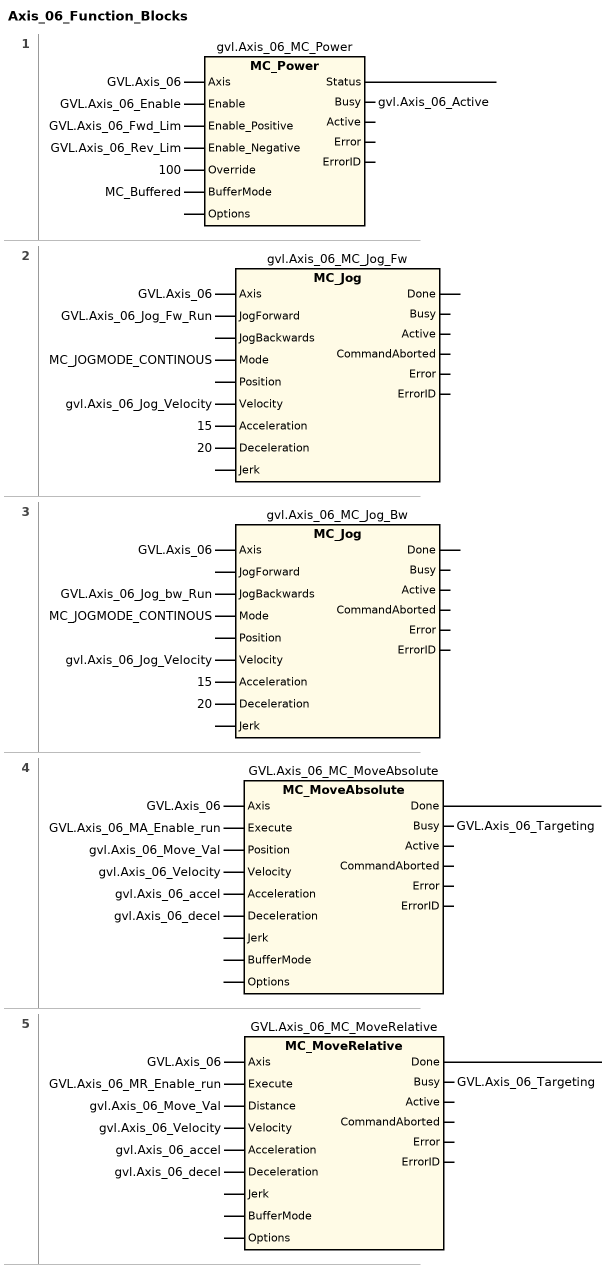
// NETWORK 1
gvl.Axis_06_MC_Power(
    Axis := GVL.Axis_06,
    Enable := GVL.Axis_06_Enable,
    Enable_Positive := GVL.Axis_06_Fwd_Lim,
    Enable_Negative := GVL.Axis_06_Rev_Lim,
    Override := 100,
    BufferMode := MC_Buffered,
    Busy => gvl.Axis_06_Active); // MC_Power

// NETWORK 2
gvl.Axis_06_MC_Jog_Fw(
    Axis := GVL.Axis_06,
    JogForward := GVL.Axis_06_Jog_Fw_Run,
    Mode := MC_JOGMODE_CONTINOUS,
    Velocity := gvl.Axis_06_Jog_Velocity,
    Acceleration := 15,
    Deceleration := 20); // MC_Jog

// NETWORK 3
gvl.Axis_06_MC_Jog_Bw(
    Axis := GVL.Axis_06,
    JogBackwards := GVL.Axis_06_Jog_bw_Run,
    Mode := MC_JOGMODE_CONTINOUS,
    Velocity := gvl.Axis_06_Jog_Velocity,
    Acceleration := 15,
    Deceleration := 20); // MC_Jog

// NETWORK 4
GVL.Axis_06_MC_MoveAbsolute(
    Axis := GVL.Axis_06,
    Execute := GVL.Axis_06_MA_Enable_run,
    Position := gvl.Axis_06_Move_Val,
    Velocity := gvl.Axis_06_Velocity,
    Acceleration := gvl.Axis_06_accel,
    Deceleration := gvl.Axis_06_decel,
    Busy => GVL.Axis_06_Targeting); // MC_MoveAbsolute

// NETWORK 5
GVL.Axis_06_MC_MoveRelative(
    Axis := GVL.Axis_06,
    Execute := GVL.Axis_06_MR_Enable_run,
    Distance := gvl.Axis_06_Move_Val,
    Velocity := gvl.Axis_06_Velocity,
    Acceleration := gvl.Axis_06_accel,
    Deceleration := gvl.Axis_06_decel,
    Busy => GVL.Axis_06_Targeting); // MC_MoveRelative

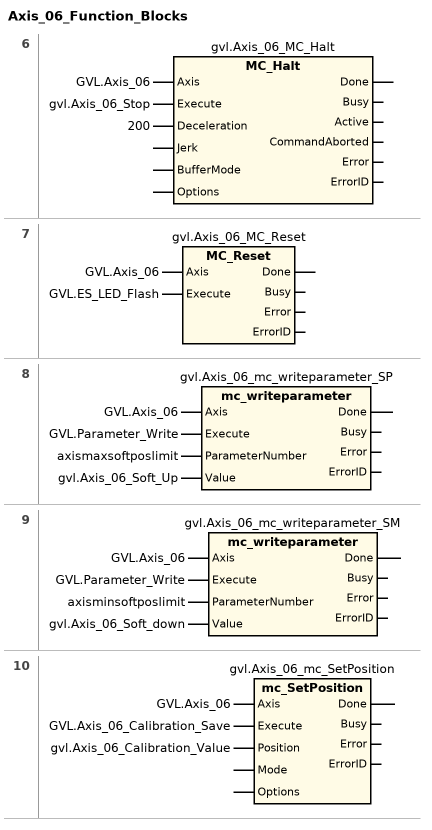
// NETWORK 6
gvl.Axis_06_MC_Halt(Axis := GVL.Axis_06, Execute := gvl.Axis_06_Stop, Deceleration := 200); // MC_Halt

// NETWORK 7
gvl.Axis_06_MC_Reset(Axis := GVL.Axis_06, Execute := GVL.ES_LED_Flash); // MC_Reset

// NETWORK 8
gvl.Axis_06_mc_writeparameter_SP(
    Axis := GVL.Axis_06,
    Execute := GVL.Parameter_Write,
    ParameterNumber := axismaxsoftposlimit,
    Value := gvl.Axis_06_Soft_Up); // mc_writeparameter

// NETWORK 9
gvl.Axis_06_mc_writeparameter_SM(
    Axis := GVL.Axis_06,
    Execute := GVL.Parameter_Write,
    ParameterNumber := axisminsoftposlimit,
    Value := gvl.Axis_06_Soft_down); // mc_writeparameter

// NETWORK 10
gvl.Axis_06_mc_SetPosition(
    Axis := GVL.Axis_06,
    Execute := GVL.Axis_06_Calibration_Save,
    Position := gvl.Axis_06_Calibration_Value); // mc_SetPosition

END_PROGRAM

// ---- POUs/Axis_06_Logic.TcPOU
PROGRAM Axis_06_Logic
VAR
	TON_0: TON;
	TON_1: TON;
	TON_2: TON;
	TON_3: TON;
	Axis_06_Velocity_Range: LREAL;
	Axis_06_Velocity_Scale: LREAL;
	Axis_06_Velocity_Raw: LREAL;
	Axis_06_Soft_Range: LREAL;
	Axis_06_Soft_Position: LREAL;
	Axis_06_Soft_Position_In_Range: LREAL;
END_VAR

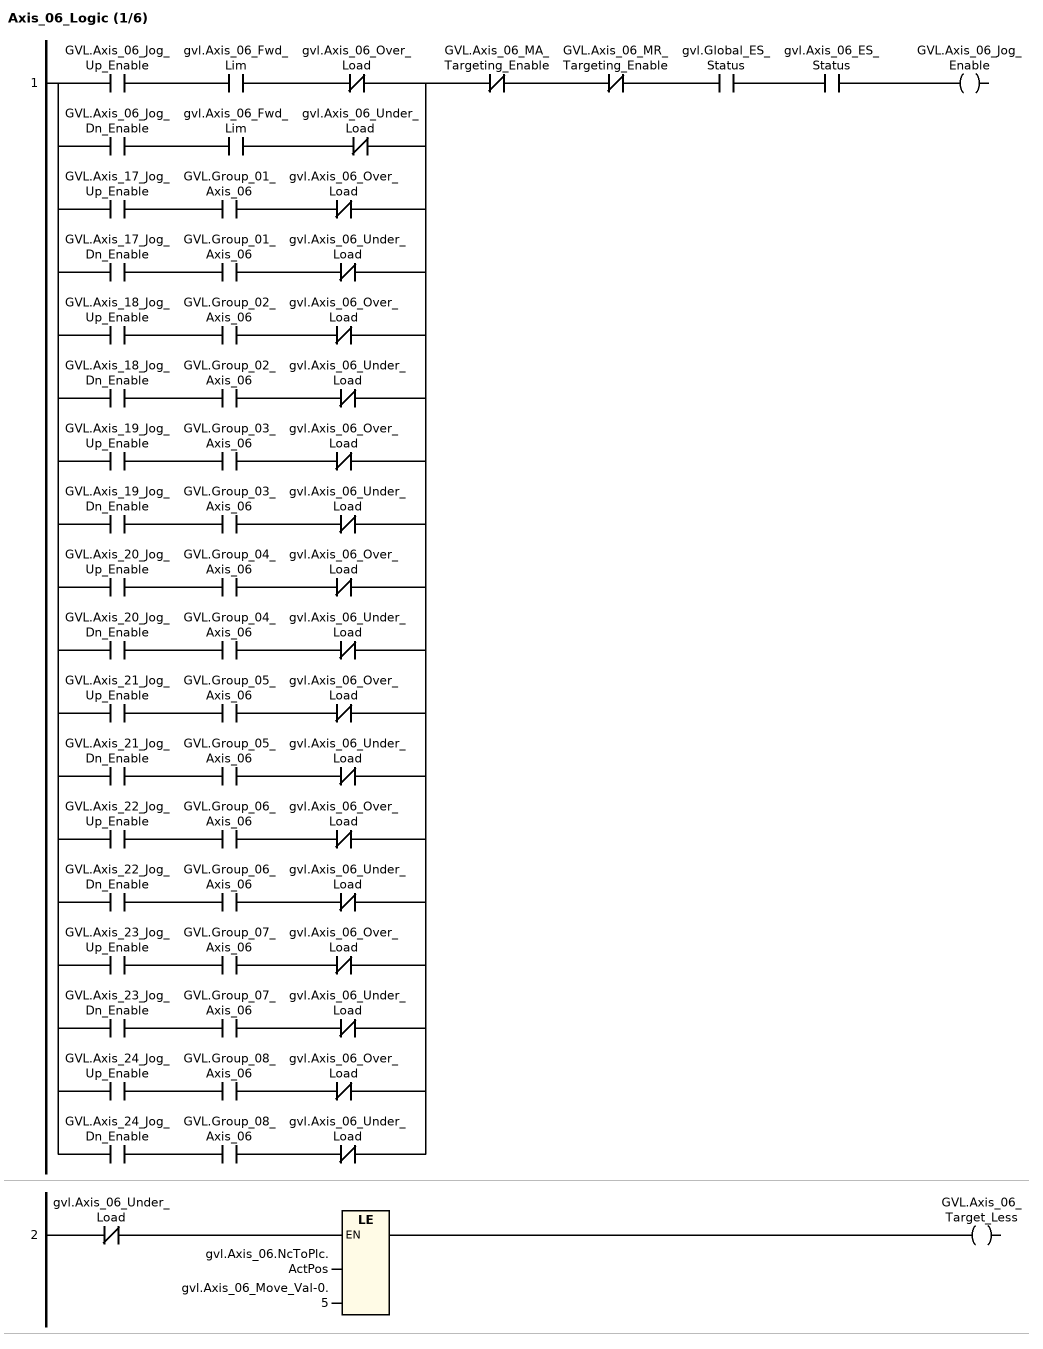
// NETWORK 1
GVL.Axis_06_Jog_Enable := (GVL.Axis_06_Jog_Up_Enable AND gvl.Axis_06_Fwd_Lim AND NOT gvl.Axis_06_Over_Load OR GVL.Axis_06_Jog_Dn_Enable AND gvl.Axis_06_Fwd_Lim AND NOT gvl.Axis_06_Under_Load OR GVL.Axis_17_Jog_Up_Enable AND GVL.Group_01_Axis_06 AND NOT gvl.Axis_06_Over_Load OR GVL.Axis_17_Jog_Dn_Enable AND GVL.Group_01_Axis_06 AND NOT gvl.Axis_06_Under_Load OR GVL.Axis_18_Jog_Up_Enable AND GVL.Group_02_Axis_06 AND NOT gvl.Axis_06_Over_Load OR GVL.Axis_18_Jog_Dn_Enable AND GVL.Group_02_Axis_06 AND NOT gvl.Axis_06_Under_Load OR GVL.Axis_19_Jog_Up_Enable AND GVL.Group_03_Axis_06 AND NOT gvl.Axis_06_Over_Load OR GVL.Axis_19_Jog_Dn_Enable AND GVL.Group_03_Axis_06 AND NOT gvl.Axis_06_Under_Load OR GVL.Axis_20_Jog_Up_Enable AND GVL.Group_04_Axis_06 AND NOT gvl.Axis_06_Over_Load OR GVL.Axis_20_Jog_Dn_Enable AND GVL.Group_04_Axis_06 AND NOT gvl.Axis_06_Under_Load OR GVL.Axis_21_Jog_Up_Enable AND GVL.Group_05_Axis_06 AND NOT gvl.Axis_06_Over_Load OR GVL.Axis_21_Jog_Dn_Enable AND GVL.Group_05_Axis_06 AND NOT gvl.Axis_06_Under_Load OR GVL.Axis_22_Jog_Up_Enable AND GVL.Group_06_Axis_06 AND NOT gvl.Axis_06_Over_Load OR GVL.Axis_22_Jog_Dn_Enable AND GVL.Group_06_Axis_06 AND NOT gvl.Axis_06_Under_Load OR GVL.Axis_23_Jog_Up_Enable AND GVL.Group_07_Axis_06 AND NOT gvl.Axis_06_Over_Load OR GVL.Axis_23_Jog_Dn_Enable AND GVL.Group_07_Axis_06 AND NOT gvl.Axis_06_Under_Load OR GVL.Axis_24_Jog_Up_Enable AND GVL.Group_08_Axis_06 AND NOT gvl.Axis_06_Over_Load OR GVL.Axis_24_Jog_Dn_Enable AND GVL.Group_08_Axis_06 AND NOT gvl.Axis_06_Under_Load) AND NOT GVL.Axis_06_MA_Targeting_Enable AND NOT GVL.Axis_06_MR_Targeting_Enable AND gvl.Global_ES_Status AND gvl.Axis_06_ES_Status;

// NETWORK 2
GVL.Axis_06_Target_Less := NOT gvl.Axis_06_Under_Load AND gvl.Axis_06.NcToPlc.ActPos <= (gvl.Axis_06_Move_Val-0.5);

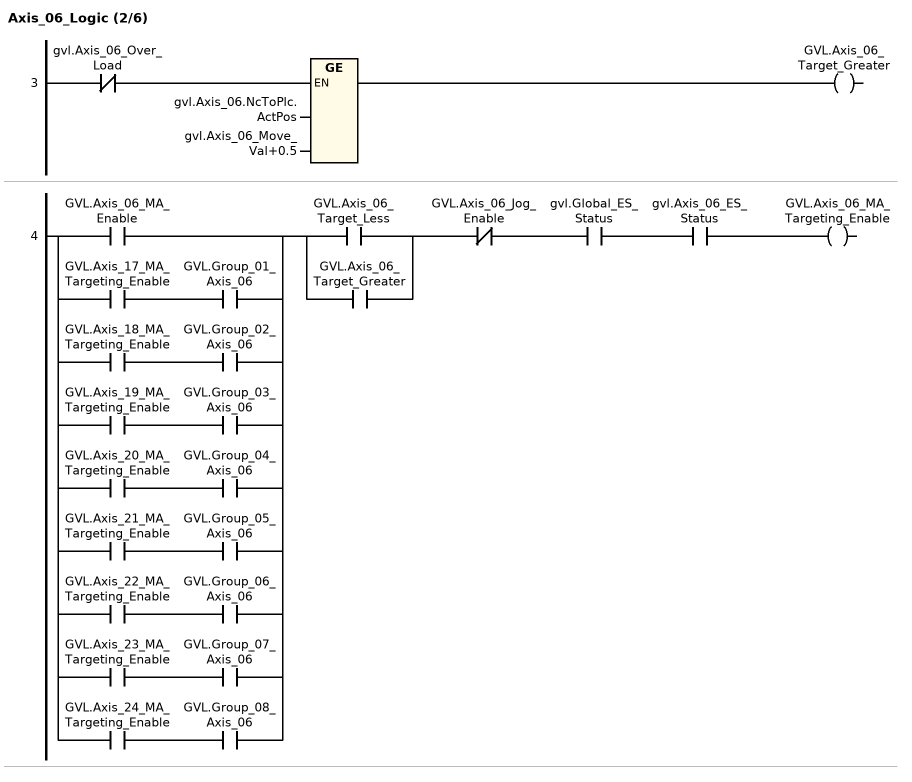
// NETWORK 3
GVL.Axis_06_Target_Greater := NOT gvl.Axis_06_Over_Load AND gvl.Axis_06.NcToPlc.ActPos >= (gvl.Axis_06_Move_Val+0.5);

// NETWORK 4
GVL.Axis_06_MA_Targeting_Enable := (GVL.Axis_06_MA_Enable OR GVL.Axis_17_MA_Targeting_Enable AND GVL.Group_01_Axis_06 OR GVL.Axis_18_MA_Targeting_Enable AND GVL.Group_02_Axis_06 OR GVL.Axis_19_MA_Targeting_Enable AND GVL.Group_03_Axis_06 OR GVL.Axis_20_MA_Targeting_Enable AND GVL.Group_04_Axis_06 OR GVL.Axis_21_MA_Targeting_Enable AND GVL.Group_05_Axis_06 OR GVL.Axis_22_MA_Targeting_Enable AND GVL.Group_06_Axis_06 OR GVL.Axis_23_MA_Targeting_Enable AND GVL.Group_07_Axis_06 OR GVL.Axis_24_MA_Targeting_Enable AND GVL.Group_08_Axis_06) AND (GVL.Axis_06_Target_Less OR GVL.Axis_06_Target_Greater) AND NOT GVL.Axis_06_Jog_Enable AND gvl.Global_ES_Status AND gvl.Axis_06_ES_Status;

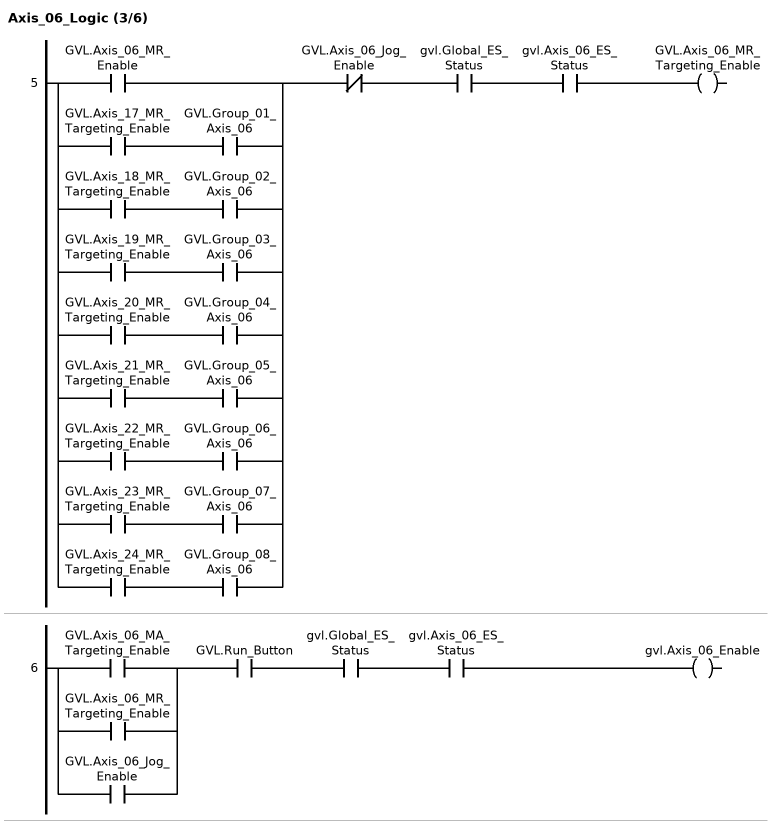
// NETWORK 5
GVL.Axis_06_MR_Targeting_Enable := (GVL.Axis_06_MR_Enable OR GVL.Axis_17_MR_Targeting_Enable AND GVL.Group_01_Axis_06 OR GVL.Axis_18_MR_Targeting_Enable AND GVL.Group_02_Axis_06 OR GVL.Axis_19_MR_Targeting_Enable AND GVL.Group_03_Axis_06 OR GVL.Axis_20_MR_Targeting_Enable AND GVL.Group_04_Axis_06 OR GVL.Axis_21_MR_Targeting_Enable AND GVL.Group_05_Axis_06 OR GVL.Axis_22_MR_Targeting_Enable AND GVL.Group_06_Axis_06 OR GVL.Axis_23_MR_Targeting_Enable AND GVL.Group_07_Axis_06 OR GVL.Axis_24_MR_Targeting_Enable AND GVL.Group_08_Axis_06) AND NOT GVL.Axis_06_Jog_Enable AND gvl.Global_ES_Status AND gvl.Axis_06_ES_Status;

// NETWORK 6
gvl.Axis_06_Enable := (GVL.Axis_06_MA_Targeting_Enable OR GVL.Axis_06_MR_Targeting_Enable OR GVL.Axis_06_Jog_Enable) AND GVL.Run_Button AND gvl.Global_ES_Status AND gvl.Axis_06_ES_Status;

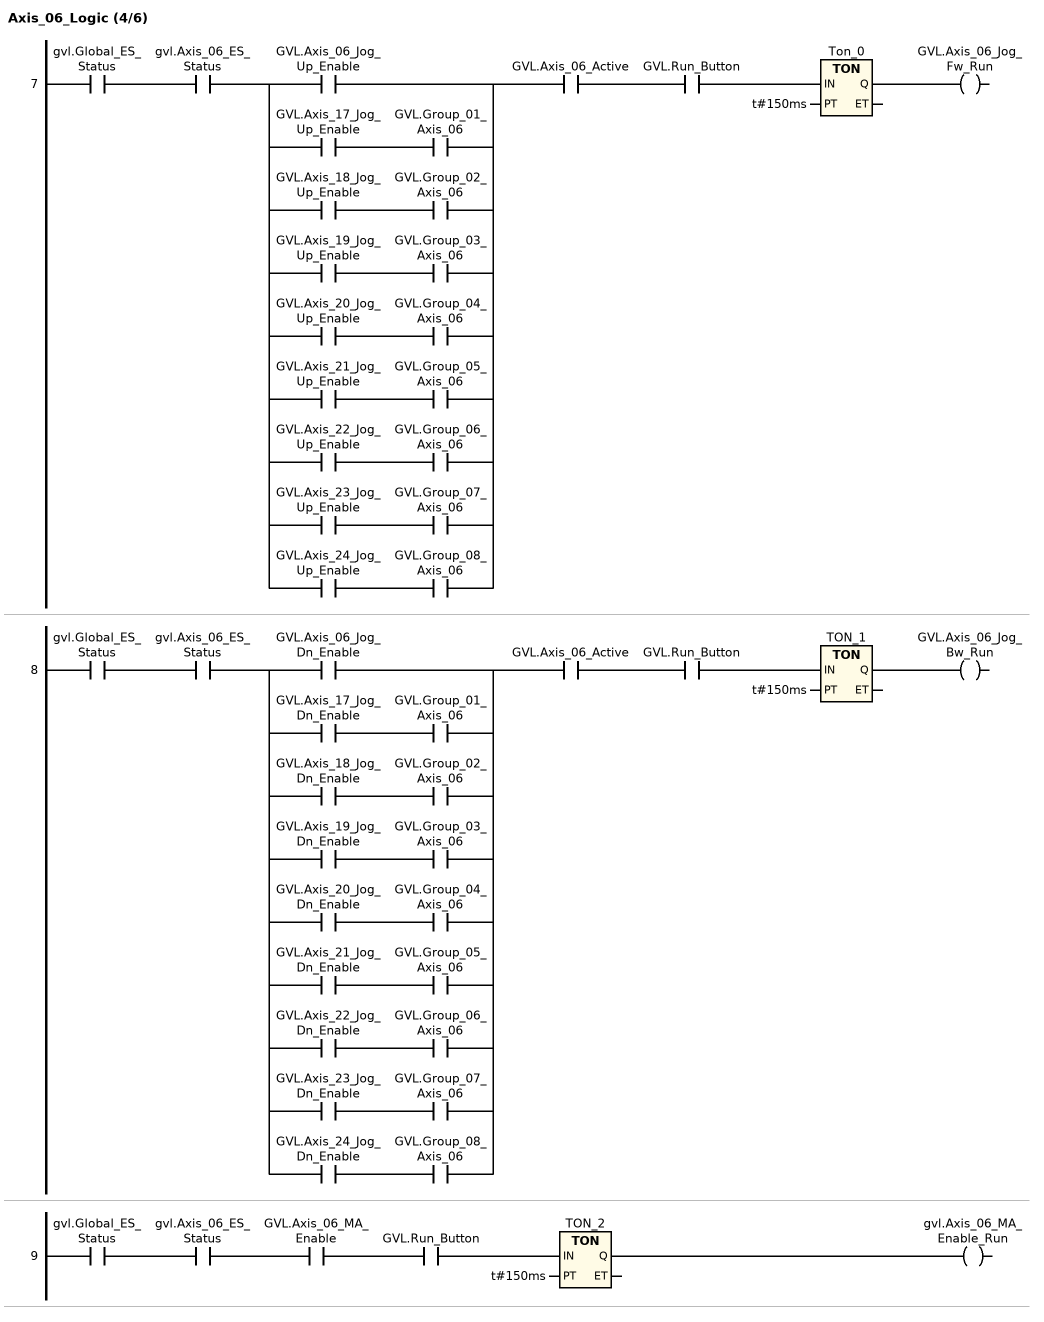
// NETWORK 7
Ton_0(IN := gvl.Global_ES_Status AND gvl.Axis_06_ES_Status AND (GVL.Axis_06_Jog_Up_Enable OR GVL.Axis_17_Jog_Up_Enable AND GVL.Group_01_Axis_06 OR GVL.Axis_18_Jog_Up_Enable AND GVL.Group_02_Axis_06 OR GVL.Axis_19_Jog_Up_Enable AND GVL.Group_03_Axis_06 OR GVL.Axis_20_Jog_Up_Enable AND GVL.Group_04_Axis_06 OR GVL.Axis_21_Jog_Up_Enable AND GVL.Group_05_Axis_06 OR GVL.Axis_22_Jog_Up_Enable AND GVL.Group_06_Axis_06 OR GVL.Axis_23_Jog_Up_Enable AND GVL.Group_07_Axis_06 OR GVL.Axis_24_Jog_Up_Enable AND GVL.Group_08_Axis_06) AND GVL.Axis_06_Active AND GVL.Run_Button, PT := t#150ms); // TON
GVL.Axis_06_Jog_Fw_Run := Ton_0.Q;

// NETWORK 8
TON_1(IN := gvl.Global_ES_Status AND gvl.Axis_06_ES_Status AND (GVL.Axis_06_Jog_Dn_Enable OR GVL.Axis_17_Jog_Dn_Enable AND GVL.Group_01_Axis_06 OR GVL.Axis_18_Jog_Dn_Enable AND GVL.Group_02_Axis_06 OR GVL.Axis_19_Jog_Dn_Enable AND GVL.Group_03_Axis_06 OR GVL.Axis_20_Jog_Dn_Enable AND GVL.Group_04_Axis_06 OR GVL.Axis_21_Jog_Dn_Enable AND GVL.Group_05_Axis_06 OR GVL.Axis_22_Jog_Dn_Enable AND GVL.Group_06_Axis_06 OR GVL.Axis_23_Jog_Dn_Enable AND GVL.Group_07_Axis_06 OR GVL.Axis_24_Jog_Dn_Enable AND GVL.Group_08_Axis_06) AND GVL.Axis_06_Active AND GVL.Run_Button, PT := t#150ms); // TON
GVL.Axis_06_Jog_Bw_Run := TON_1.Q;

// NETWORK 9
TON_2(IN := gvl.Global_ES_Status AND gvl.Axis_06_ES_Status AND GVL.Axis_06_MA_Enable AND GVL.Run_Button, PT := t#150ms); // TON
gvl.Axis_06_MA_Enable_Run := TON_2.Q;

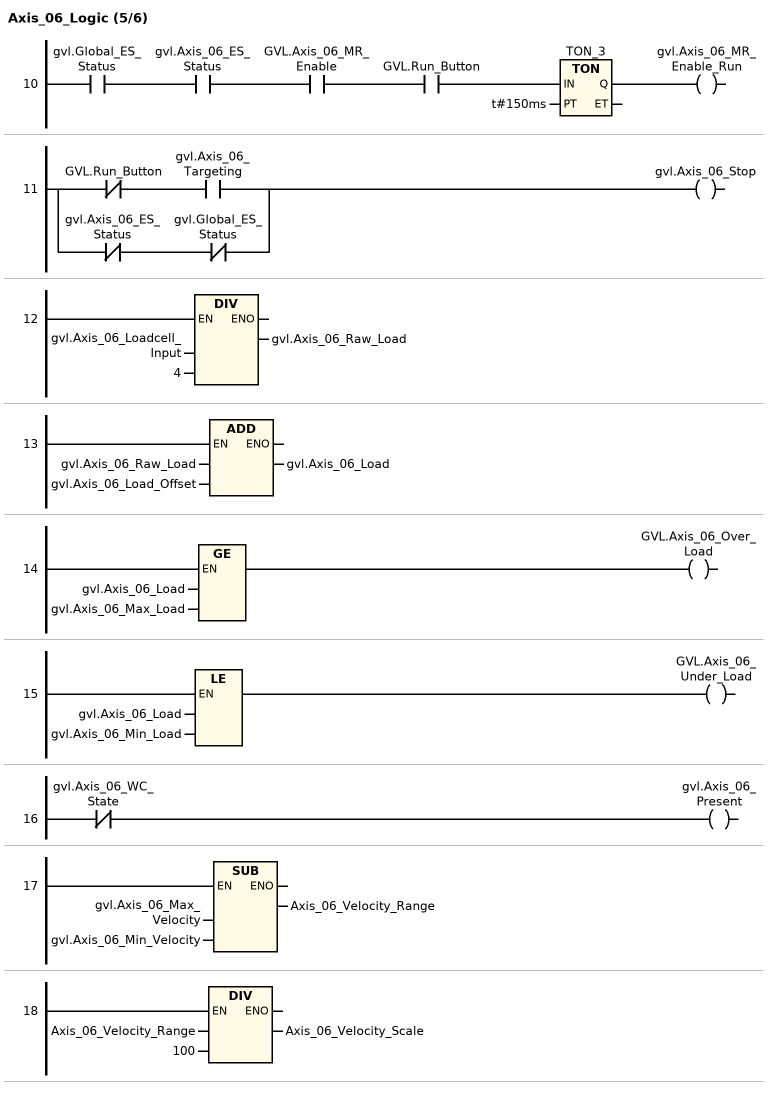
// NETWORK 10
TON_3(IN := gvl.Global_ES_Status AND gvl.Axis_06_ES_Status AND GVL.Axis_06_MR_Enable AND GVL.Run_Button, PT := t#150ms); // TON
gvl.Axis_06_MR_Enable_Run := TON_3.Q;

// NETWORK 11
gvl.Axis_06_Stop := NOT GVL.Run_Button AND gvl.Axis_06_Targeting OR NOT gvl.Axis_06_ES_Status AND NOT gvl.Global_ES_Status;

// NETWORK 12
gvl.Axis_06_Raw_Load := gvl.Axis_06_Loadcell_Input / 4;

// NETWORK 13
gvl.Axis_06_Load := gvl.Axis_06_Raw_Load + gvl.Axis_06_Load_Offset;

// NETWORK 14
GVL.Axis_06_Over_Load := gvl.Axis_06_Load >= gvl.Axis_06_Max_Load;

// NETWORK 15
GVL.Axis_06_Under_Load := gvl.Axis_06_Load <= gvl.Axis_06_Min_Load;

// NETWORK 16
gvl.Axis_06_Present := NOT gvl.Axis_06_WC_State;

// NETWORK 17
Axis_06_Velocity_Range := gvl.Axis_06_Max_Velocity - gvl.Axis_06_Min_Velocity;

// NETWORK 18
Axis_06_Velocity_Scale := Axis_06_Velocity_Range / 100;

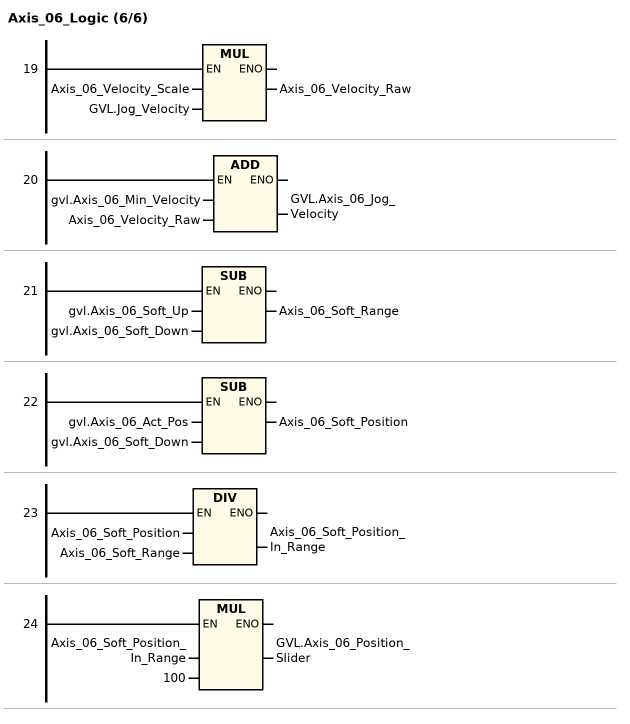
// NETWORK 19
Axis_06_Velocity_Raw := Axis_06_Velocity_Scale * GVL.Jog_Velocity;

// NETWORK 20
GVL.Axis_06_Jog_Velocity := gvl.Axis_06_Min_Velocity + Axis_06_Velocity_Raw;

// NETWORK 21
Axis_06_Soft_Range := gvl.Axis_06_Soft_Up - gvl.Axis_06_Soft_Down;

// NETWORK 22
Axis_06_Soft_Position := gvl.Axis_06_Act_Pos - gvl.Axis_06_Soft_Down;

// NETWORK 23
Axis_06_Soft_Position_In_Range := Axis_06_Soft_Position / Axis_06_Soft_Range;

// NETWORK 24
GVL.Axis_06_Position_Slider := Axis_06_Soft_Position_In_Range * 100;

END_PROGRAM

// ---- POUs/Axis_07_Function_Blocks.TcPOU
PROGRAM Axis_07_Function_Blocks
VAR
END_VAR

